FUNCTION TryConvert_REAL_TO_TIME : BOOL
VAR_INPUT
	in : REAL;
	out : REFERENCE TO TIME;
END_VAR

IF in > DatatypeLimits.MAX_VALUE_OF_REAL_WHICH_CAN_BE_HELD_IN_A_TIME THEN
	RETURN;
END_IF

IF in < DatatypeLimits.MIN_VALUE_OF_REAL_WHICH_CAN_BE_HELD_IN_A_TIME THEN
	RETURN;
END_IF

out := REAL_TO_TIME(in);
TryConvert_REAL_TO_TIME := TRUE;

END_FUNCTION

(* stored: Version 1.1.0.1, ProductVersion 3.1.4024.12
   POU TryConvert_REAL_TO_TIME: Id {382b2418-bc7d-4981-88c7-70aa7c0634b9}, SpecialFunc None *)
